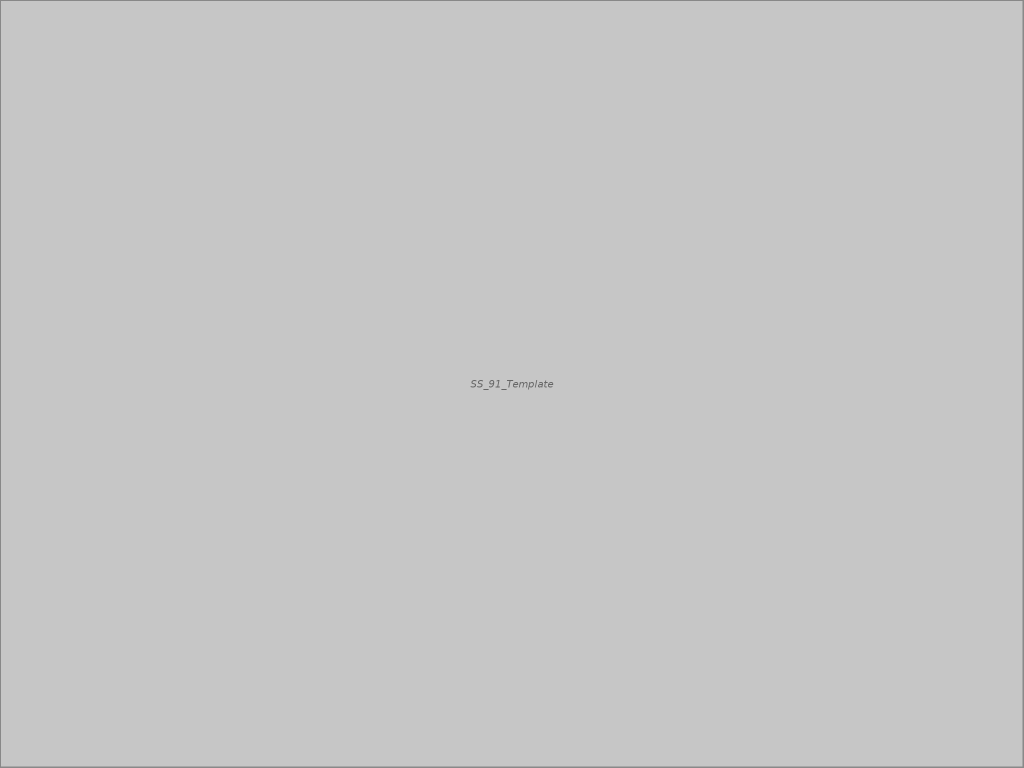
VISUALIZATION SS_12_MachineLayout  // 1024x768
    Frame (0,0 1024x768)
        shows SS_91_Template(header := gHMIData.hmiHeader)
END_VISUALIZATION

(* stored: Version 1.1.0.1, ProductVersion 3.1.4024.12
   Visu SS_12_MachineLayout: Id {88ee6430-3b99-476f-997c-dbe82955d6bd} *)
